TYPE NETWORK_BUFFER_SHORT :
STRUCT
	SIZE : UINT;
	BUFFER : NW_BUF_SHORT;
END_STRUCT
END_TYPE

(* stored: Version 1.1.0.1, ProductVersion 3.1.4024.9
   DUT NETWORK_BUFFER_SHORT: Id {5ce83c30-48af-414b-99bb-3d5d962f1e94} *)
